// TIA Portal project "PWM_MODULU_KULLANMA" (V18)

(* hardware
DEVICE "S7-1200 station_1"  S7-1200 Station
   slot 0: "Rack_0"  S7-1200 Rack  Rack  V1.0
   slot 1: "PLC_1"  CPU 1214C DC/DC/DC  6ES7 214-1AG40-0XB0  V4.6
*)

// ===== PLC "PLC_1"  CPU 1214C DC/DC/DC =====

VAR_GLOBAL   // PLC tag table "Default tag table"
   "Tag_1" AT %I0.0 : Bool;
   "Tag_2" AT %MW4 : Word;
   "Tag_3" AT %M3.0 : Bool;
   "Tag_4" AT %IW1000 : Word;
   "Tag_5" AT %MW40 : Word;
END_VAR

ORGANIZATION_BLOCK "Main"   // OB1, LAD, ProgramCycle
TITLE = "Main Program Sweep (Cycle)"
{ S7_Optimized_Access := 'TRUE' }
VERSION : 0.1
   VAR_INPUT
      Initial_Call : Bool;   // Initial call of this OB
      Remanence : Bool;   // =True, if remanent data are available
   END_VAR
BEGIN

REGION Network 1
   // 265 değeri pwm ayarlarından yazılır
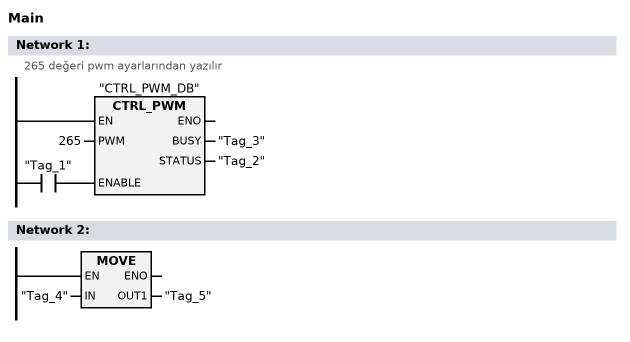
   "CTRL_PWM_DB"(PWM := 265, ENABLE := "Tag_1", BUSY => "Tag_3", STATUS => "Tag_2");   // CTRL_PWM
END_REGION

REGION Network 2
   RUNG wire#powerrail
      Move(in := "Tag_4", out1 => "Tag_5")
   END_RUNG
   // the same network as SCL:
   "Tag_5" := "Tag_4";
END_REGION
END_ORGANIZATION_BLOCK